PROGRAM main
VAR
	MODBEE_HW_INPUTS0 : MODBEE_HW_INPUTS;
	MODBEE_HW_OUTPUTS0 : MODBEE_HW_OUTPUTS;
	start : bool;
	stop : bool;
	run : bool;
	TON0 : TON;
	TON1 : TON;
	TON1_DONE : bool;
	TON0_DONE : bool;
	MODBEE_READ0 : MODBEE_READ;
	MODBEE_WRITE0 : MODBEE_WRITE;
	MBEE_READ_COILS_DONE : bool;
	MBEE_DI01 : bool;
	MBEE_DI02 : bool;
	MBEE_DI03 : bool;
	MBEE_DI04 : bool;
	MBEE_DI05 : bool;
	MBEE_DI06 : bool;
	MBEE_DI07 : bool;
	MBEE_DI08 : bool;
	MBEE_WRITE_COILS_DONE : bool;
	MBEE_DO01 : bool;
	MBEE_DO02 : bool;
	MBEE_DO03 : bool;
	MBEE_DO04 : bool;
	MBEE_DO05 : bool;
	MBEE_DO06 : bool;
	MBEE_DO07 : bool;
	MBEE_DO08 : bool;
	MODBEE_CONFIG0 : MODBEE_CONFIG;
	MODBEE_READ1 : MODBEE_READ;
	MODBEE_WRITE1 : MODBEE_WRITE;
	MBEE_AI01 : int;
	MBEE_AI02 : int;
	MBEE_AI03 : int;
	MBEE_AI04 : int;
	MBEE_AO01 : real;
	MBEE_AO02 : real;
	MBEE_AO01_TEMP : int;
	MBEE_AO02_TEMP : int;
	MODBEE_HAT_PWR0 : MODBEE_HAT_PWR;
END_VAR

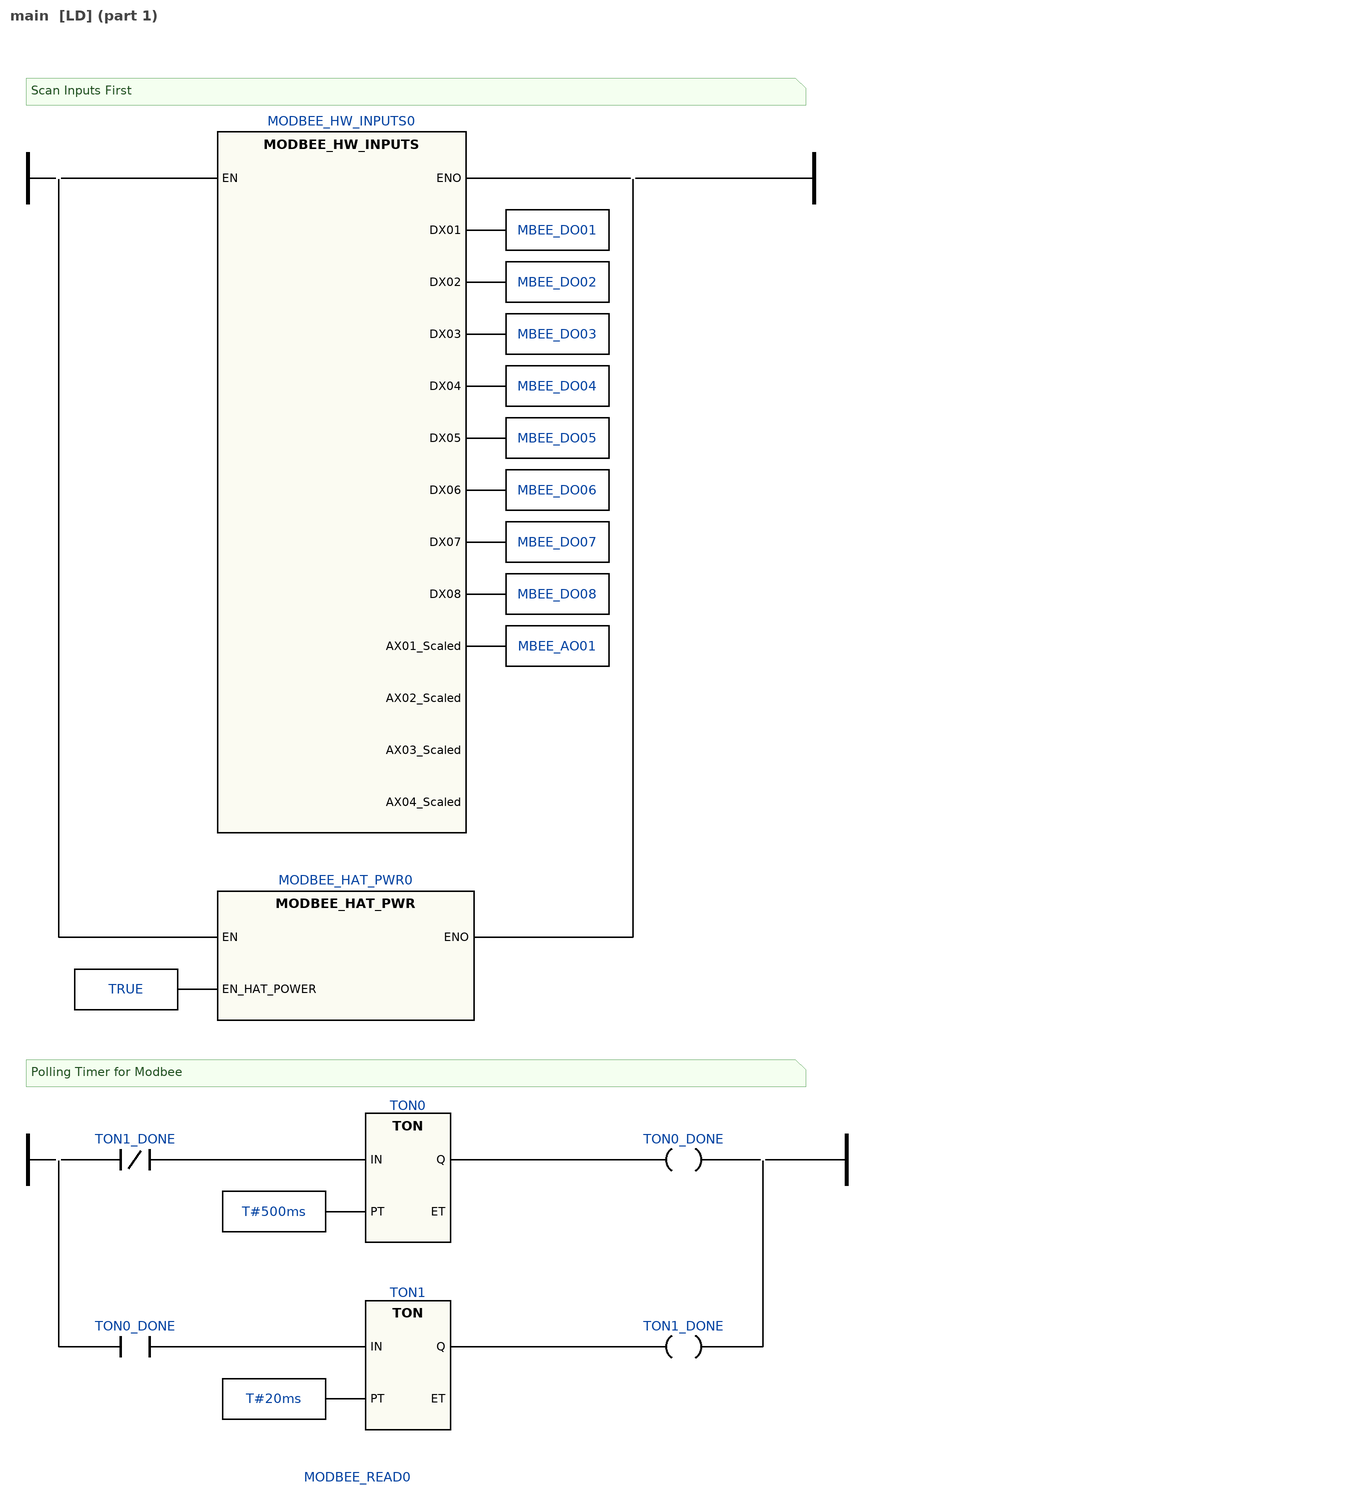
(* LD diagram, written out as Structured Text *)
(* Scan Inputs First *)
MODBEE_HW_INPUTS0();
MBEE_DO01 := MODBEE_HW_INPUTS0.DX01;
MBEE_DO02 := MODBEE_HW_INPUTS0.DX02;
MBEE_DO03 := MODBEE_HW_INPUTS0.DX03;
MBEE_DO04 := MODBEE_HW_INPUTS0.DX04;
MBEE_DO05 := MODBEE_HW_INPUTS0.DX05;
MBEE_DO06 := MODBEE_HW_INPUTS0.DX06;
MBEE_DO07 := MODBEE_HW_INPUTS0.DX07;
MBEE_DO08 := MODBEE_HW_INPUTS0.DX08;
MBEE_AO01 := MODBEE_HW_INPUTS0.AX01_Scaled;
(* Polling Timer for Modbee *)
TON0(IN := NOT TON1_DONE, PT := T#500ms);
TON0_DONE := TON0.Q;
TON1(IN := TON0_DONE, PT := T#20ms);
TON1_DONE := TON1.Q;
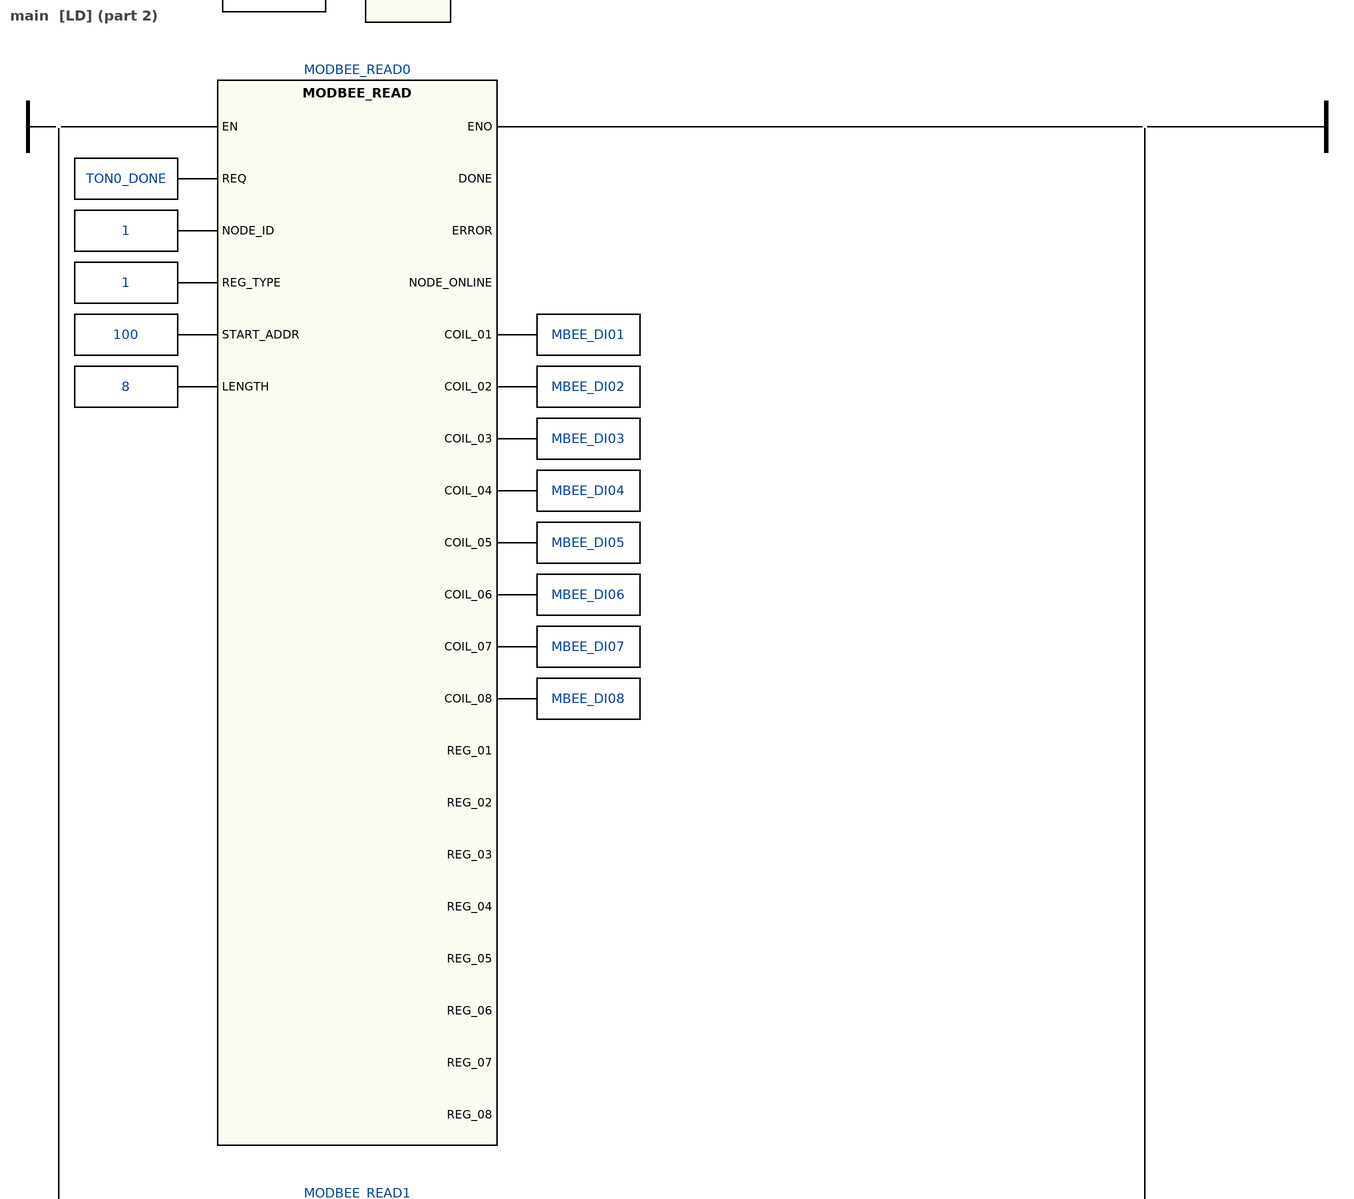
MODBEE_READ0(REQ := TON0_DONE, NODE_ID := 1, REG_TYPE := 1, START_ADDR := 100, LENGTH := 8);
MBEE_DI01 := MODBEE_READ0.COIL_01;
MBEE_DI02 := MODBEE_READ0.COIL_02;
MBEE_DI03 := MODBEE_READ0.COIL_03;
MBEE_DI04 := MODBEE_READ0.COIL_04;
MBEE_DI05 := MODBEE_READ0.COIL_05;
MBEE_DI06 := MODBEE_READ0.COIL_06;
MBEE_DI07 := MODBEE_READ0.COIL_07;
MBEE_DI08 := MODBEE_READ0.COIL_08;
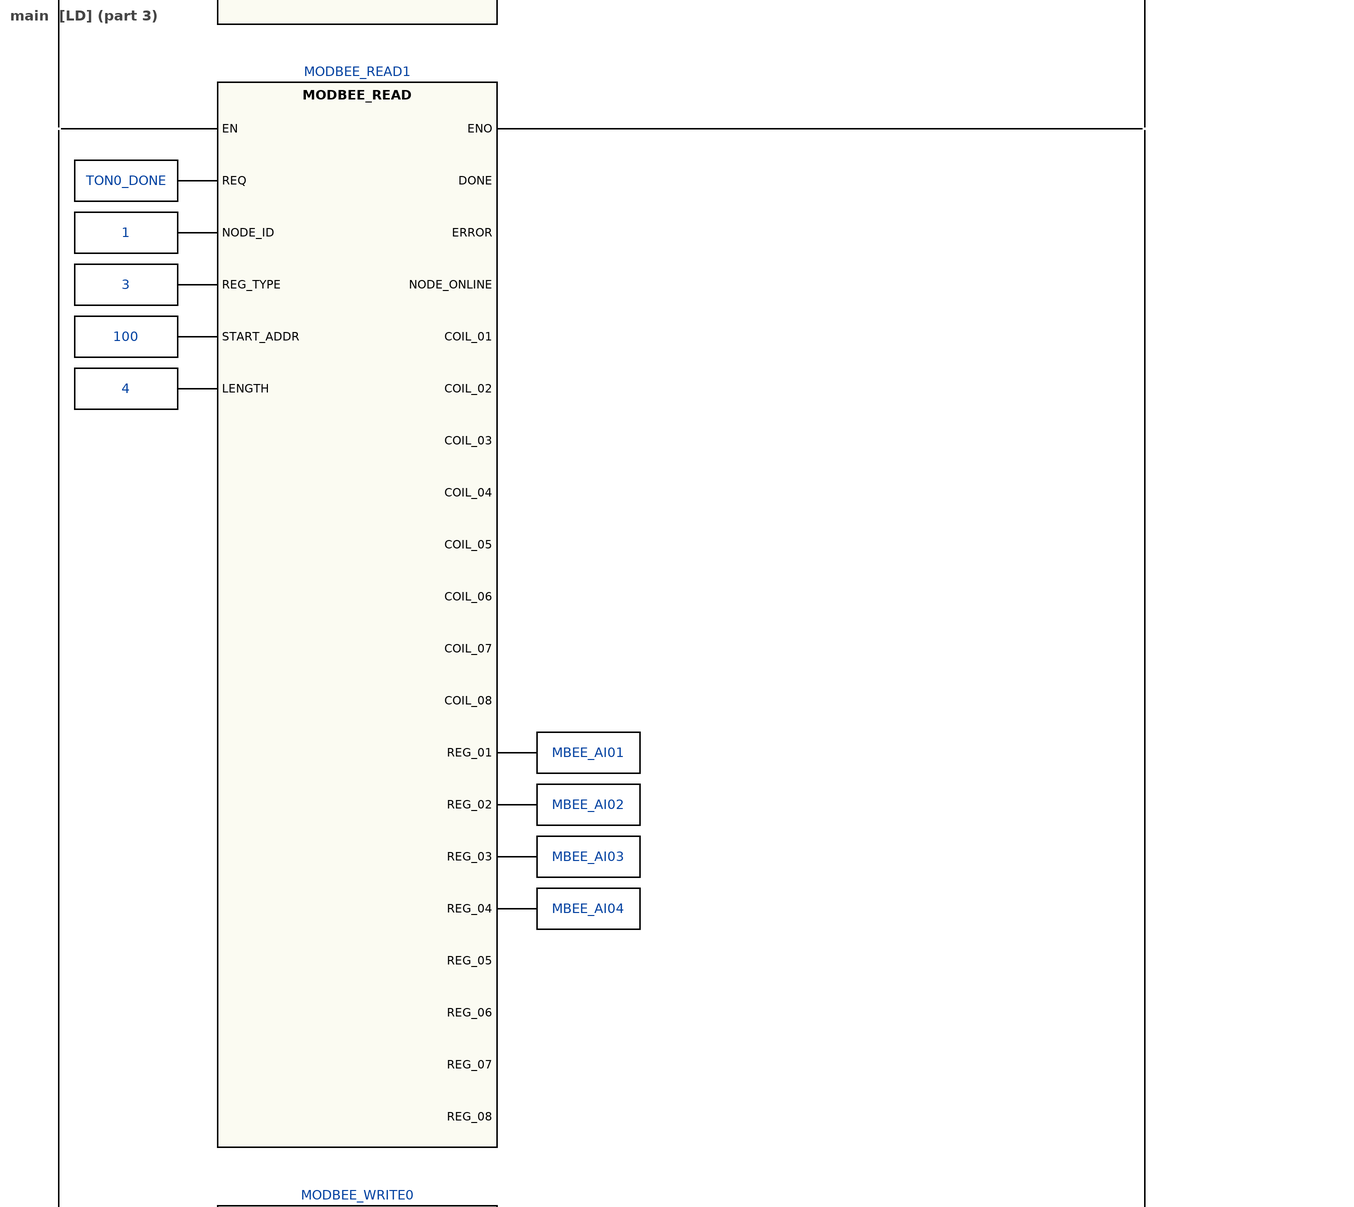
MODBEE_READ1(REQ := TON0_DONE, NODE_ID := 1, REG_TYPE := 3, START_ADDR := 100, LENGTH := 4);
MBEE_AI01 := MODBEE_READ1.REG_01;
MBEE_AI02 := MODBEE_READ1.REG_02;
MBEE_AI03 := MODBEE_READ1.REG_03;
MBEE_AI04 := MODBEE_READ1.REG_04;
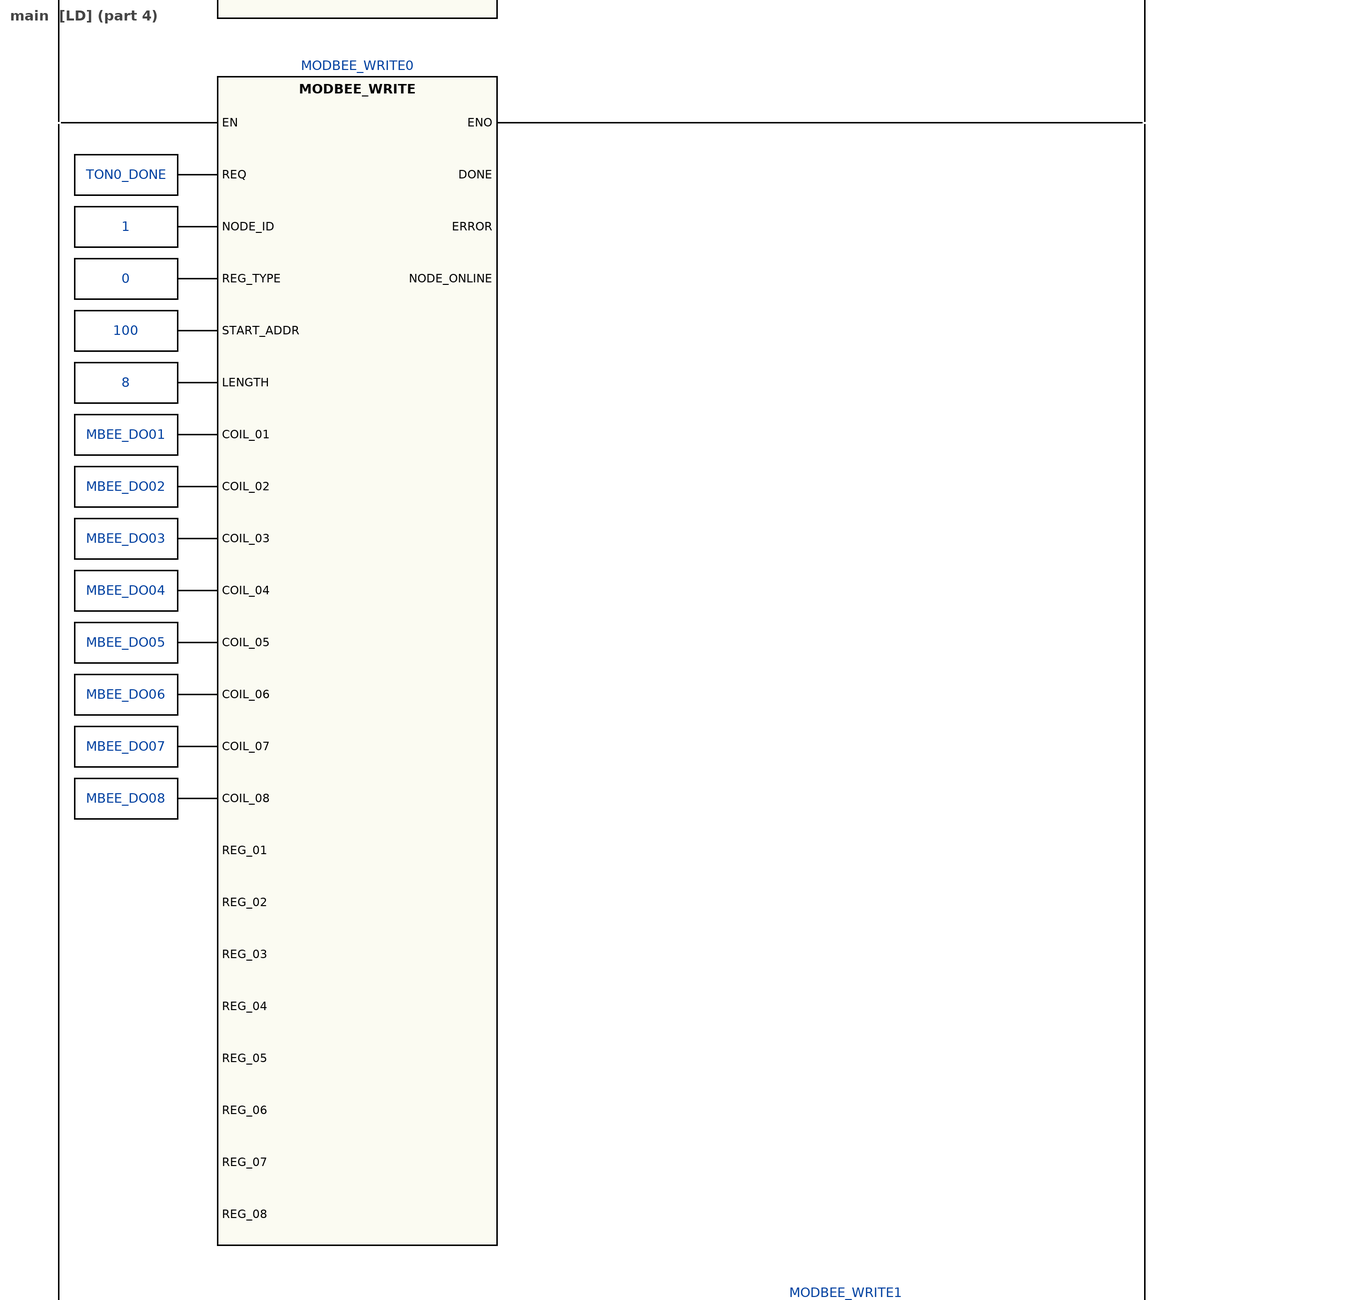
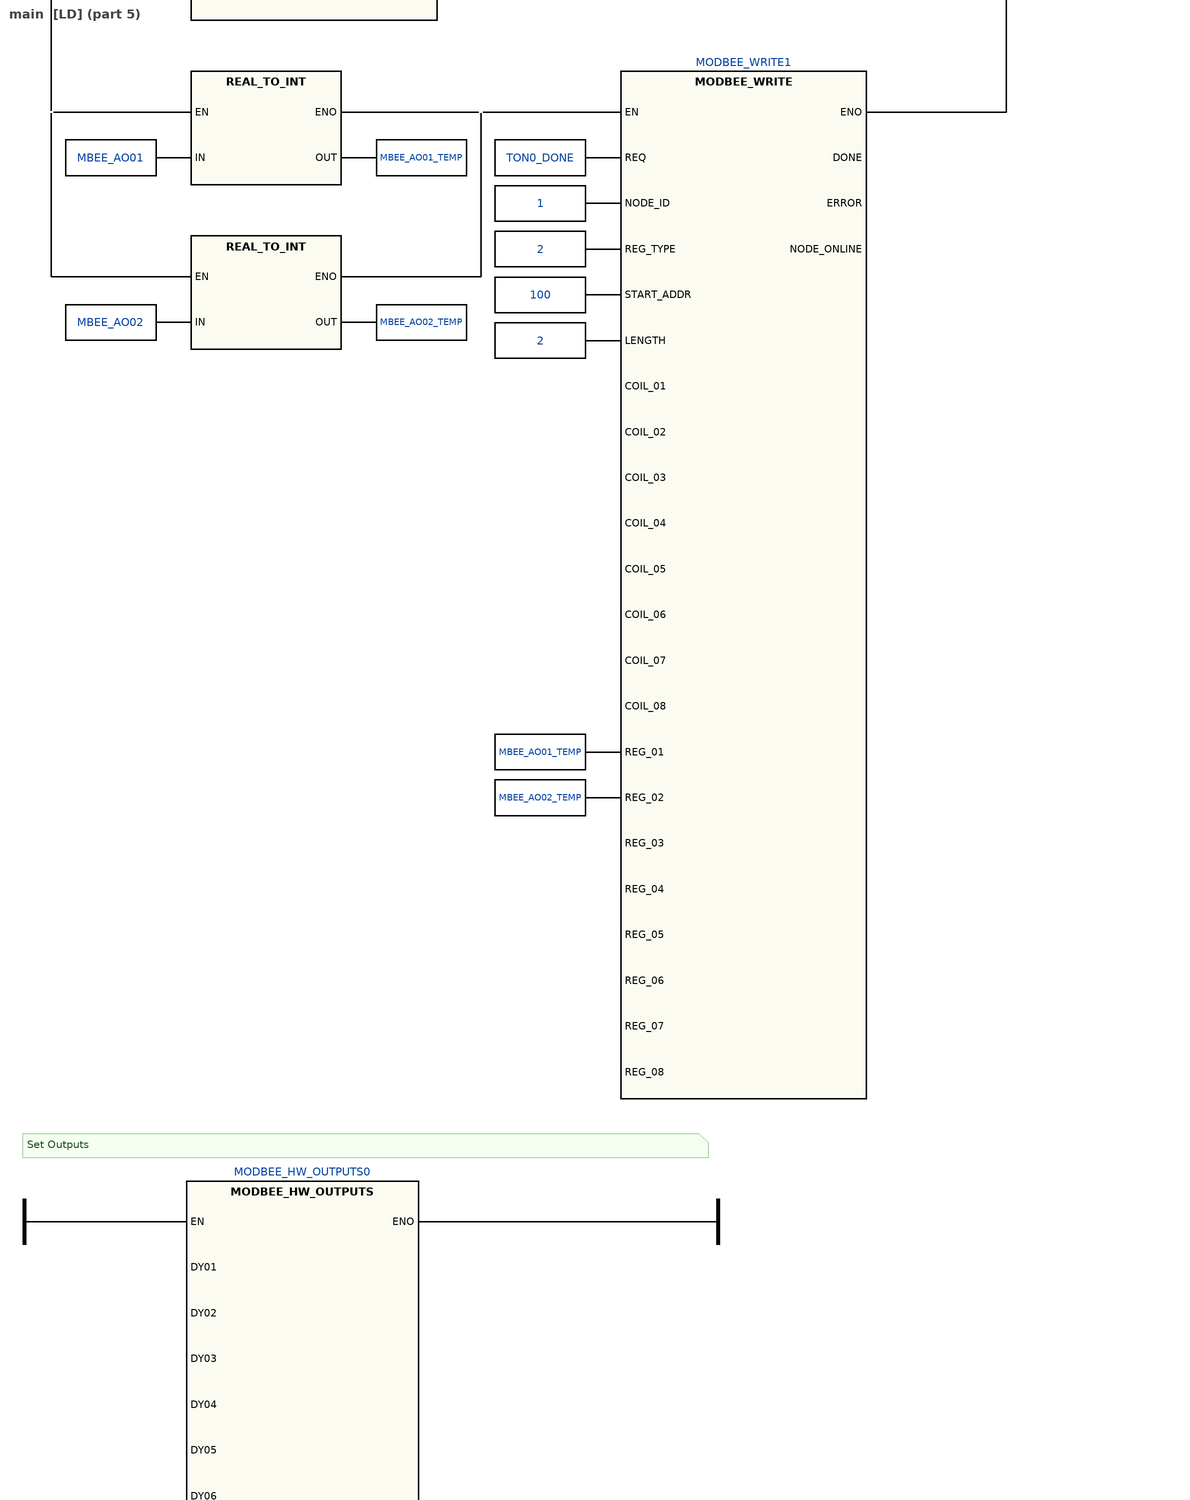
MBEE_AO01_TEMP := REAL_TO_INT(MBEE_AO01);
MBEE_AO02_TEMP := REAL_TO_INT(MBEE_AO02);
MODBEE_HAT_PWR0(EN_HAT_POWER := TRUE);
MODBEE_WRITE0(REQ := TON0_DONE, NODE_ID := 1, REG_TYPE := 0, START_ADDR := 100, LENGTH := 8, COIL_01 := MBEE_DO01, COIL_02 := MBEE_DO02, COIL_03 := MBEE_DO03, COIL_04 := MBEE_DO04, COIL_05 := MBEE_DO05, COIL_06 := MBEE_DO06, COIL_07 := MBEE_DO07, COIL_08 := MBEE_DO08);
MODBEE_WRITE1(REQ := TON0_DONE, NODE_ID := 1, REG_TYPE := 2, START_ADDR := 100, LENGTH := 2, REG_01 := MBEE_AO01_TEMP, REG_02 := MBEE_AO02_TEMP);
(* Set Outputs *)
MODBEE_HW_OUTPUTS0();
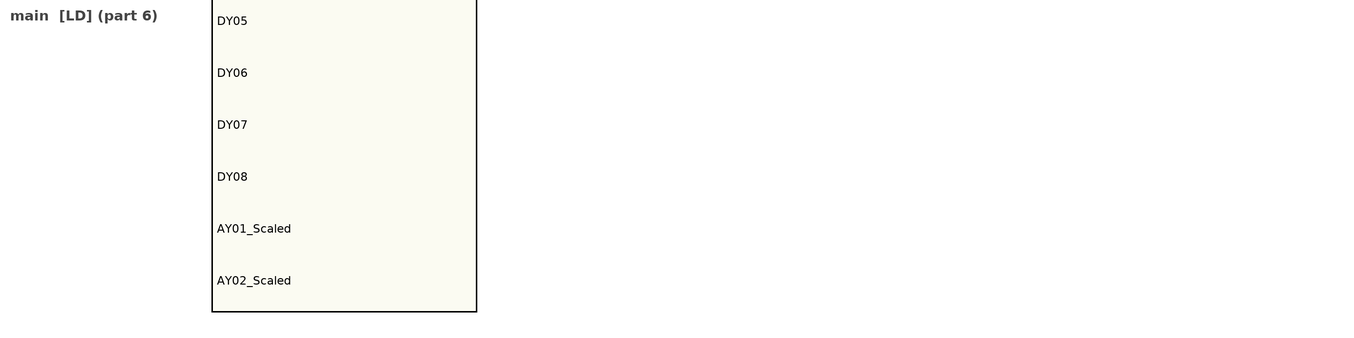
END_PROGRAM
